// TIA Portal V17 export
// export: Created 2025-03-07T09:19:56.8772606Z, ExportSetting WithDefaults, DisplayName Totally Integrated Automation Portal, DisplayVersion V17 Update 8, DisplayName TIA Portal Openness, DisplayVersion V17 Update 8, DisplayName TIA Portal Version Control Interface, DisplayVersion V17, DisplayName SINAMICS Startdrive Advanced, DisplayVersion V17 SP2, DisplayName SINAMICS Startdrive G110M, G120, G120C, G120D, G120P, G115D, DisplayVersion V17 SP2, DisplayName SINAMICS Startdrive G130, G150, S120, S150, SINAMICS MV, S210, DisplayVersion V17 SP2, DisplayName STEP 7 Professional, DisplayVersion V17 Update 8, DisplayName SINUMERIK ONE STEP 7 Toolbox, DisplayVersion V17 Update 12, DisplayName SINUMERIK 840D sl STEP 7 Toolbox, DisplayVersion V17 Update 12, DisplayName STEP 7 Safety, DisplayVersion V17 Update 6, DisplayName WinCC Advanced, DisplayVersion V17 Update 8
TYPE "LASER ACTIVE"
// stored: IsFailsafeCompliant false
   STRUCT
      "EMISSION LASER STILL PERMANENT CONDITIONS" : Bool;
      "EMISSION LASER STILL ENABLE REQUEST" : Bool;
      "EMISSION LASER STILL DISABLE REQUEST" : Bool;
      "EMISSION LASER STILL ENABLE MODE" : Bool;
      "LASER ACTIVE A" : Bool;
      "LASER ACTIVE START GENERAL CONDITIONS" : Bool;
      "LASER ACTIVE START INITIAL CONDITIONS" : Bool;
      "LASER ACTIVE MANUAL START REQUEST" : Bool;
      "LASER ACTIVE AUTO START REQUEST" : Bool;
      "LASER ACTIVE START REQUEST" : Bool;
      "LASER ACTIVE START COMMAND" : Bool;
      "LASER ACTIVE LASER ACTIVE ON" : Bool;
      "LASER ACTIVE FEEDBACK ON" : Bool;
      "LASER ACTIVE STOP GENERAL CONDITIONS" : Bool;
      "LASER ACTIVE STOP INITIAL CONDITIONS" : Bool;
      "LASER ACTIVE MANUAL STOP REQUEST" : Bool;
      "LASER ACTIVE AUTO STOP REQUEST" : Bool;
      "LASER ACTIVE STOP REQUEST" : Bool;
      "LASER ACTIVE STOP COMMAND" : Bool;
      "LASER ACTIVE STOPPED" : Bool;
      "LASER ACTIVE FEEDBACK OFF" : Bool;
      "LASER ACTIVE PROGRAM NOT ACTIVE" : Bool;
      "LASER ACTIVE WARNING GONE" : Bool;
      "LASER ACTIVE START GENERAL CONDITION HELP" : Bool;
      "LASER ACTIVE START INITIAL CONDITION HELP" : Bool;
      "LASER ACTIVE STOP GENERAL CONDITION HELP" : Bool;
      "LASER ACTIVE STOP INITIAL CONDITION HELP" : Bool;
      "LASER ACTIVE FAULT" : Bool;
   END_STRUCT;
END_TYPE
